FUNCTION_BLOCK E_MERGE_3 (* Merge (OR) of three input events (generic FB) *)
  (* Standard: 61499-1 Annex A; Function: Output EO is triggered when either EI1 or EI2 is received; Description: Copyright (c) 2017, 2025 fortiss GmbH, HR Agrartechnik GmbH This program and the accompanying materials are made available under the terms of the Eclipse Public License 2.0 which is available at https://www.eclipse.org/legal/epl-2.0/ SPDX-License-Identifier: EPL-2.0 *)
  (* Version 3.0, 2025-04-14, Patrick Aigner, changed package *)
  (* Version 1.1, 2025-02-12, Franz H??pfinger, HR Agrartechnik GmbH, copy from E_MERGE and make a E_MERGE3 in the same way *)
  (* Version 1.0, 2017, Alois Zoitl, fortiss GmbH, initial API and implementation and/or initial documentation *)
  PACKAGE iec61499::events;
  {SET_ATTRIBUTE(eclipse4diac::core::GenericClassName, 'GEN_E_MERGE')}
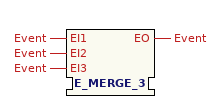
  EVENT_INPUT
    EI1; (* First input event *)
    EI2; (* Second input event *)
    EI3; (* Third input event *)
  END_EVENT
  EVENT_OUTPUT
    EO; (* Output Event *)
  END_EVENT
END_FUNCTION_BLOCK
